TYPE (* logiBUS AI Struct Dual *)
  (* Version 1.0, 2026-05-28, franz *)
  PACKAGE logiBUS::io::AI;
  IMPORT logiBUS::io::AI::logiBUS_AI_S;
  logiBUS_AI_S_Dual : STRUCT
    Up : logiBUS_AI_S := (Pin := 255); (* forward, up, right, clockwise *)
    Down : logiBUS_AI_S := (Pin := 255); (* backward, down, left, counter-clockwise *)
  END_STRUCT;
END_TYPE
